(* IEC 61131-3 sources: CODESYS-IO-Visualization/CODESYS-IO-Visualization.fbsproj/Subs/IO, 10 files *)

(* ---- CodeSysCPU.prg.st ---- *)
PROGRAM CodeSysCPU

VAR_IN_OUT
	cpu: CodeSysCPU_UDT;
END_VAR

IF (cpu.PersistSize = 0) THEN
	cpu.PersistSize := SIZEOF(CodeSysCPU_UDT);
END_IF;

IF (cpu.Init OR cpu.AppResult <> 0) THEN
	cpu.App := AppGetCurrent(pResult := ADR(cpu.AppResult));
	IF (cpu.App <> 0) AND(cpu.AppResult = 0) THEN
		cpu.AppInfo := AppGetApplicationInfo(pApp := cpu.App, pResult := ADR(cpu.AppInfoResult));
		IF (cpu.AppInfo <> 0) AND (cpu.AppInfoResult = 0) THEN
 			cpu.AppProjectName := TO_WSTRING(cpu.AppInfo^.pstProjectName^);
 			cpu.AppAuthor := TO_WSTRING(cpu.AppInfo^.pstAuthor^);
 			cpu.AppVersion := TO_WSTRING(cpu.AppInfo^.pstVersion^);
 			cpu.AppDescription := TO_WSTRING(cpu.AppInfo^.pstDescription^);
 			cpu.AppProfile := TO_WSTRING(cpu.AppInfo^.pstProfile^);

			GetDateYear(Clock := DT_TO_DATE(cpu.AppInfo^.dtLastChanges), value => cpu.AppLastChange.Year);
			GetDateMonth(Clock := DT_TO_DATE(cpu.AppInfo^.dtLastChanges), value => cpu.AppLastChange.Month);
			GetDayOfMonth(Clock := DT_TO_DATE(cpu.AppInfo^.dtLastChanges), value => cpu.AppLastChange.Day);
			GetDTHour(Clock := cpu.AppInfo^.dtLastChanges, value => cpu.AppLastChange.Hour);
			GetDTMinute(Clock := cpu.AppInfo^.dtLastChanges, value => cpu.AppLastChange.Minute);
			GetDTSecond(Clock := cpu.AppInfo^.dtLastChanges, value => cpu.AppLastChange.Second);
			cpu.AppLastChange.DateTimeString := DateTimeStampToString(DateTimeStamp := cpu.AppLastChange);
		END_IF;
	END_IF;
	cpu.Init := FALSE;
END_IF;

CycleTime(value := cpu.CT);
cpu.SampleSeconds := cpu.SampleSeconds + cpu.CT.Sec;

// only read memory and cpu data every 10 seconds
IF (cpu.SampleSeconds < 10.0) THEN
	RETURN;
END_IF;

cpu.SampleSeconds := 0.0;

// Get CPU Info - Raspberry Pi ONLY - requires Shell Access enabled in /etc/codesyscontrol/CODESYSControl_User.cfg file
// Add
//	[SysProcess]
//  Command=AllowAll
ReadCPUDetails();

cpu.CpuUsage := ReadCPUDetails.cpuUsage;
cpu.Temperature := ReadCPUDetails.cpuTemp;
cpu.MemFree := ReadCPUDetails.memFree;
cpu.MemFree_MB := ReadCPUDetails.memFree_MB;
cpu.memTotal := ReadCPUDetails.memTotal;
cpu.memTotal_MB := ReadCPUDetails.memTotal_MB;
cpu.memUsed := ReadCPUDetails.memUsed;
cpu.memUsed_MB := ReadCPUDetails.memUsed_MB;

(* ---- IO_Simulator.prg.st ---- *)
__METADATA__
{
  "v3Meta": {
    "objectGuid": "030a1301-75cd-4f4e-867e-5d1ddb7f8ba8",
    "objectTypeGuid": "6f9dac99-8de1-4efc-8465-68ac443b7d08",
    "embeddedObjectTypeGuids": [
      "a9ed5b7e-75c5-4651-af16-d2c27e98cb94",
      "3b83b776-fb25-43b8-99f2-3c507c9143fc"
    ],
    "properties": {},
    "subObjects": {}
  }
}
__DECLARATION__
PROGRAM IO_Simulator
VAR_IN_OUT
	Data: IO_Simulator_UDT;
END_VAR
__IMPLEMENTATION__
Data.RandomNumber := OSCAT_BASIC.RDM(Data.RandomNumber);
Data.Noise := Data.RandomNumber * Data.irNoisePct;

Data.ChangeRamp(
	X := Data.irPercent,
	A_UP := Data.irChangeRate,
	A_DN := Data.irChangeRate * -1,
	VU_MAX := Data.irChangeRate,
	VD_MAX := Data.irChangeRate * -1,
	LIMIT_LOW := 0.0,
	LIMIT_HIGH := 100.0
);

IF (NOT Data.ibDisableOutput) THEN
	Data.orPercent := Data.Noise + Data.ChangeRamp.Y;
	Data.obValue := Data.ibValue;
END_IF;

Data.orValue := Data.irLowLimit + ((Data.orPercent / 100.0) * (Data.irHighLimit - Data.irLowLimit));

(* ---- IOA_Input.prg.st ---- *)
PROGRAM IOA_Input

VAR_IN_OUT
	Data: Channel_UDT;
END_VAR

VAR_INPUT
	ModuleStatus: DINT;
	ModuleCI: BOOL;
END_VAR

IF (Data.CI OR ModuleCI) THEN
	Data.StatusString := "Control Inhibited";
	Data.StatusCode := -1;
ELSE
	IF (Data.SimulationEnable AND Simulation.SimulationEnable) THEN
		ModuleStatus := 0;
		Data.ValueStatus := 0;
		Data.StatusCode := Data.Simulator.odiStatusCode;
		Data.StatusString := Data.Simulator.osStatusCode;
	ELSE
		IF (ModuleStatus > 0) THEN
			Data.StatusCode := ModuleStatus;
			Data.StatusString := "Module Failed, check Module Status";
		ELSE
			Data.StatusCode := WORD_TO_DINT(Data.ValueStatus);
			IO_StatusCodeToString(Data := Data);
		END_IF;
	END_IF;
END_IF;

Data.Invalid.Value := (Data.StatusCode > 0);
AlarmDigital(alarm := Data.Invalid);

IF (NOT FPU.IsRealNaN(Data.ValueRawAnalog)) THEN
	IF (Data.ValueRawAnalog > (Data.ZeroRaw + (Data.SpanRaw * 1.04))) THEN
		Data.ValueRawAnalog := Data.ZeroRaw + Data.SpanRaw;
	END_IF;

	IF (Data.ValueRawAnalog < (Data.ZeroRaw - (Data.SpanRaw * 0.04))) THEN
		Data.ValueRawAnalog := Data.ZeroRaw;
	END_IF;
END_IF;

IF (NOT Data.CI) AND (NOT ModuleCI) THEN
	IF (Data.SimulationEnable AND Simulation.SimulationEnable) THEN
		IO_Simulator(Data := Data.Simulator);
		Data.ValueEu := Data.Simulator.orValue;
	ELSE
		IF (NOT FPU.IsRealNaN(Data.ValueRawAnalog)) THEN
			IF (Data.SpanRaw <> 0.0) THEN
				Data.ValueEu := Data.ZeroEu + (((Data.ValueRawAnalog - Data.ZeroRaw) / Data.SpanRaw) * Data.SpanEu);
			ELSE
				Data.ValueEu := 0.0;
			END_IF;
		ELSE
			Data.ValueEu := 0.0;
		END_IF;
	END_IF;
END_IF;

IF (NOT FPU.IsRealNaN(Data.ValueRawAnalog)) THEN
	IF (Data.SpanEu <> 0.0) THEN
		Data.ValuePct := ((Data.ValueEu - Data.ZeroEu) / Data.SpanEu) * 100.0;
		IF (Data.ValuePct > 100.0) THEN
			Data.ValuePct := 100.0;
		END_IF;
		IF (Data.ValuePct < 0.0) THEN
			Data.ValuePct := 0.0;
		END_IF;
	ELSE
		Data.ValuePct := 0.0;
	END_IF;
ELSE
	Data.ValuePct := 0.0;
END_IF;

(* ---- IOA_Output.prg.st ---- *)
PROGRAM IOA_Output

VAR_IN_OUT
	Data: Channel_UDT;
END_VAR

VAR_INPUT
	ModuleStatus: DINT;
	ModuleCI: BOOL;
END_VAR

IF (Data.CI OR ModuleCI) THEN
	Data.StatusString := "Control Inhibited";
	Data.StatusCode := -1;
ELSE
	IF (ModuleStatus  > 0) THEN
		Data.StatusCode := ModuleStatus;
		Data.StatusString := "Module Failed, check Module Status";
	ELSE
		Data.StatusCode := WORD_TO_DINT(Data.ValueStatus);
		IO_StatusCodeToString(Data := Data);
	END_IF;
END_IF;

Data.Invalid.Value := (Data.StatusCode > 0);
AlarmDigital(alarm := Data.Invalid);

IF (NOT Data.CI) AND (NOT ModuleCI) THEN
	IF (Data.SpanEu <> 0.0) THEN
		Data.ValueRawAnalogOut := Data.ZeroRaw + (((Data.ValueEu - Data.ZeroEu) / Data.SpanEu) * Data.SpanRaw);
	ELSE
		Data.ValueRawAnalogOut := 0.0;
	END_IF;

	IF (Data.ValueRawAnalogOut > (Data.ZeroRaw + (Data.SpanRaw * 1.04))) THEN
		Data.ValueRawAnalogOut := Data.ZeroRaw + Data.SpanRaw;
	END_IF;

	IF (Data.ValueRawAnalogOut < (Data.ZeroRaw - (Data.SpanRaw * 0.04))) THEN
		Data.ValueRawAnalogOut := Data.ZeroRaw;
	END_IF;
END_IF;

IF (Data.SpanEu <> 0.0) THEN
	Data.ValuePct := ((Data.ValueEu - Data.ZeroEu) / Data.SpanEu) * 100.0;
	IF (Data.ValuePct > 100.0) THEN
		Data.ValuePct := 100.0;
	END_IF;
	IF (Data.ValuePct < 0.0) THEN
		Data.ValuePct := 0.0;
	END_IF;
ELSE
	Data.ValuePct := 0.0;
END_IF;

(* ---- IOD_Input.prg.st ---- *)
PROGRAM IOD_Input

VAR_IN_OUT
	Data: Channel_UDT;
END_VAR

VAR_INPUT
	ModuleStatus: DINT;
	ModuleCI: BOOL;
END_VAR

IF (Data.CI OR ModuleCI) THEN
	Data.StatusString := "Control Inhibited";
	Data.StatusCode := -1;
ELSE
	IF (Data.SimulationEnable AND Simulation.SimulationEnable) THEN
		ModuleStatus := 0;
		Data.ValueStatus := 0;
		Data.StatusCode := Data.Simulator.odiStatusCode;
		Data.StatusString := Data.Simulator.osStatusCode;
	ELSE
		IF (ModuleStatus > 0) THEN
			Data.StatusCode := ModuleStatus;
			Data.StatusString := "Module Failed, check Module Status";
		ELSE
			Data.StatusCode := WORD_TO_DINT(Data.ValueStatus);
			IO_StatusCodeToString(Data := Data);
		END_IF;
	END_IF;
END_IF;

Data.Invalid.Value := (Data.StatusCode > 0);
AlarmDigital(alarm := Data.Invalid);

IF (NOT Data.CI) AND (NOT ModuleCI) THEN
	IF (Data.InvertValue) THEN
		IF (Data.SimulationEnable AND Simulation.SimulationEnable) THEN
			IO_Simulator(Data := Data.Simulator);
			Data.ValueDig := (NOT Data.Simulator.obValue);
		ELSE
			Data.ValueDig := (NOT Data.ValueRawDigital);
		END_IF;
	ELSE
		IF (Data.SimulationEnable AND Simulation.SimulationEnable) THEN
			IO_Simulator(Data := Data.Simulator);
			Data.ValueDig := Data.Simulator.obValue;
		ELSE
			Data.ValueDig := Data.ValueRawDigital;
		END_IF;
	END_IF;
END_IF;

(* ---- IOD_Output.prg.st ---- *)
PROGRAM IOD_Output

VAR_IN_OUT
	Data: Channel_UDT;
END_VAR

VAR_INPUT
	ModuleStatus: DINT;
	ModuleCI: BOOL;
END_VAR

IF (Data.CI OR ModuleCI) THEN
	Data.StatusString := "Control Inhibited";
	Data.StatusCode := -1;
ELSE
	IF (ModuleStatus > 0) THEN
		Data.StatusCode := ModuleStatus;
		Data.StatusString := "Module Failed, check Module Status";
	ELSE
		Data.StatusCode := WORD_TO_DINT(Data.ValueStatus);
		IO_StatusCodeToString(Data := Data);
	END_IF;
END_IF;

Data.Invalid.Value := (Data.StatusCode > 0);
AlarmDigital(alarm := Data.Invalid);

IF (NOT Data.CI) AND (NOT ModuleCI) THEN
	IF (Data.InvertValue) THEN
		Data.ValueRawDigitalOut := (NOT Data.ValueDig);
	ELSE
		Data.ValueRawDigitalOut := Data.ValueDig;
	END_IF;
END_IF;

(* ---- ReadCPUDetails.prg.st ---- *)
PROGRAM ReadCPUDetails
VAR
	getTempCmd : STRING := 'vcgencmd measure_temp | sed $"s/temp=//; s/$'C//$"';
 	getCPUUsageCmd : STRING := 'top -bn1 | awk $'/^%Cpu/ {printf $"%.1f\n$", $$2}$'';
 	getMemoryTotalCmd : STRING := 'free | grep -E $"Mem$" | awk $'{print $$2}$'';
 	getMemoryUsedCmd : STRING := 'free | grep -E $"Mem$" | awk $'{print $$3}$'';
 	getMemoryFreeCmd : STRING := 'free | grep -E $"Mem$" | awk $'{print $$4}$'';

	command1 : STRING;
	commandToRun: INT;	// 0 = Temp, 1 = CPU, 2 = Memory Total, 3 = Memory Used, 4 = Memory Free

	stdout : STRING(1000) := '';
	Result : RTS_IEC_RESULT;
	xExecuteSysP: BOOL;
	xshowCPUInfo: BOOL;
	done: BOOL;

	dlyTimer: Timer_UDT := (PT := 0.25);
END_VAR

VAR_OUTPUT
	cpuTemp: REAL;
	cpuUsage: REAL;
	memTotal: DINT;
	memTotal_MB: REAL;
	memUsed: DINT;
	memUsed_MB: REAL;
	memFree: DINT;
	memFree_MB: REAL;
END_VAR

//Attention: allow shell commands in CODESYSControl.cfg

CASE commandToRun OF
	0: command1 := getTempCmd;
	1: command1 := getCPUUsageCmd;
	2: command1 := getMemoryTotalCmd;
	3: command1 := getMemoryUsedCmd;
	4: command1 := getMemoryFreeCmd;
END_CASE;

dlyTimer.In := (NOT done);

Timer(TimerData := dlyTimer);

IF (dlyTimer.Q) THEN
	SysProcess.SysProcessExecuteCommand2(pszCommand:=command1, pszStdOut:=stdout, udiStdOutLen:= SIZEOF(stdout),pResult := ADR(Result));
	done := TRUE;
END_IF;

IF (done AND Result = CmpErrors.Errors.ERR_OK) THEN
	IF (LEN(stdout) > 0) THEN
		CASE commandToRun OF
			0: cpuTemp := STRING_TO_REAL(stdout);
			1: cpuUsage := STRING_TO_REAL(stdout);
			2: memTotal := STRING_TO_DINT(stdout);
			   memTotal_MB := DINT_TO_REAL(memTotal) / 1024.0;
			3: memUsed := STRING_TO_DINT(stdout);
			   memUsed_MB := DINT_TO_REAL(memUsed) / 1024.0;
			4: memFree := STRING_TO_DINT(stdout);
			   memFree_MB := DINT_TO_REAL(memFree) / 1024.0;
		END_CASE;
	END_IF;

	commandToRun := commandToRun + 1;
	IF (commandToRun > 4) THEN
		commandToRun := 0;
	END_IF;

	done := FALSE;
END_IF;

(* ---- RotorkValve.prg.st ---- *)
PROGRAM RotorkValve

VAR_IN_OUT
	Data: RotorkValve_UDT;
	InputData: RotorkValve_MBIO_InputData_UDT;
	OutputData: RotorkValve_MBIO_OutputData_UDT;
END_VAR

// Assign Input Data from either the Modbus Device or the Simulator
IF (Simulation.SimulationEnable AND Data.SimulationEnable) THEN
	RotorkValve_Simulator(Data := Data.Simulator);
	Data.InputData := Data.Simulator.InputData;
ELSE
	Data.InputData := InputData;
END_IF;

IF (NOT Data.CI) THEN
	// Output Data
	Data.OutputData.Reg05 := INT_TO_WORD(Data.Actuator_Control);
	Data.OutputData.Reg06 := REAL_TO_WORD(Data.Actuator_Position_Command * 10.0);
	Data.OutputData.Reg07 := INT_TO_WORD(Data.SignalLossAction);
	Data.OutputData.Reg13 := INT_TO_WORD(Data.SignalLossPosition);

	// Input Data
	Data.InputReg00 := Data.InputData.Reg00;
	Data.Actuator_Moving := Data.InputData.Reg00.0;
	Data.Valve_Closed := Data.InputData.Reg00.1;
	Data.Valve_Opened := Data.InputData.Reg00.2;
	Data.Running_Closed := Data.InputData.Reg00.3;
	Data.Running_Open := Data.InputData.Reg00.4;
	Data.Remote_Selected := Data.InputData.Reg00.5;
	Data.Local_Stop_Selected_Offline := Data.InputData.Reg00.6;
	Data.Local_Stop_Selected := Data.InputData.Reg00.7;
	Data.Thermostat_Tripped := Data.InputData.Reg00.8;
	Data.Monitor_Relay := Data.InputData.Reg00.9;
	Data.Valve_Obstructed := Data.InputData.Reg00.10;
	Data.Valve_Jammed := Data.InputData.Reg00.11;
	Data.Valve_Moving_By_Hand := Data.InputData.Reg00.12;
	Data.Moving_Inhibited_by_MIT := Data.InputData.Reg00.13;
	Data.Position_Control_Enabled := Data.InputData.Reg00.14;
	Data.EEPROM_Checksum_Failure := Data.InputData.Reg00.15;

	Data.InputReg01 := Data.InputData.Reg01;
	Data.Battery_Low := Data.InputData.Reg01.0;
	Data.Open_Interlock_Active := Data.InputData.Reg01.1;
	Data.Close_Interlock_Active := Data.InputData.Reg01.2;
	Data.DI_1 := Data.InputData.Reg01.3;
	Data.DI_2 := Data.InputData.Reg01.4;
	Data.DI_3 := Data.InputData.Reg01.5;
	Data.DI_4 := Data.InputData.Reg01.6;
	Data.Reserved_7 := Data.InputData.Reg01.7;
	Data.Reserved_8 := Data.InputData.Reg01.8;
	Data.Reserved_9 := Data.InputData.Reg01.9;
	Data.Control_Contention := Data.InputData.Reg01.10;
	Data.Partial_Stroke_Test_in_Progress := Data.InputData.Reg01.11;
	Data.Partial_Stroke_Test_Error := Data.InputData.Reg01.12;
	Data.General_Alarm := Data.InputData.Reg01.13;
	Data.Reserved_14 := Data.InputData.Reg01.14;
	Data.Reserved_15 := Data.InputData.Reg01.15;

	Data.Actuator_Torque := WORD_TO_REAL(Data.InputData.Reg02);
	Data.Valve_Position := WORD_TO_REAL(Data.InputData.Reg03) / 10.0;
	Data.Analog_Input := WORD_TO_REAL(Data.InputData.Reg04) / 10.0;

	// Modbus Slave Data
	Data.SlaveState := Data.InputData.State;
	Data.SlaveError := Data.InputData.Error;
	Data.SlaveErrorCode := Data.InputData.ErrorCode;

	IF (Data.SlaveState = 2) THEN
		Data.Status := INT_TO_DINT(Data.SlaveErrorCode);
	ELSE
		Data.Status := UINT_TO_DINT(Data.SlaveState) + 1000;
	END_IF;
ELSE
	Data.Status := DINT#-1;
END_IF

// Output Data
IF (Simulation.SimulationEnable AND Data.SimulationEnable) THEN
	Data.Simulator.OutputData := Data.OutputData;
ELSE
	OutputData := Data.OutputData;
END_IF;

(* ---- RotorkValve_Simulator.prg.st ---- *)
PROGRAM RotorkValve_Simulator

VAR_IN_OUT
	Data: RotorkValve_Simulator_UDT;
END_VAR

// Set Valve Data from ModbusIO
Data.ibUsePosCmd := TRUE;

// Check for Comm Fail and set the valve position based on SignalLoss settings
IF (Data.InputData.Error OR (Data.InputData.State <> 2) OR (Data.InputData.ErrorCode <> 0)) THEN
	CASE Data.OutputData.Reg07 OF
		1: Data.irPosCmd := 100.0;
		3: Data.irPosCmd := 0.0;
		5: Data.irPosCmd := Data.orPosition;
		7: Data.irPosCmd := WORD_TO_REAL(Data.OutputData.Reg13);
	END_CASE;
ELSE
	Data.irPosCmd := WORD_TO_REAL(Data.OutputData.Reg06) / 10.0;
END_IF;

Data.ibAlarm := Data.Battery_Low OR Data.Open_Interlock_Active OR Data.Close_Interlock_Active OR Data.General_Alarm;
Data.ibFault := Data.Thermostat_Tripped OR Data.Valve_Obstructed OR Data.Valve_Jammed OR Data.Moving_Inhibited_by_MIT OR Data.EEPROM_Checksum_Failure;

// Call Simulator
ValveSimulator(Data := Data);

// Set Valve Output information from simulator
Data.InputData.Reg02 := 55;
Data.InputData.Reg03 := REAL_TO_WORD(Data.orPosition * 10.0);
Data.InputData.Reg04 := REAL_TO_WORD(Data.Analog_Input * 10.0);

Data.InputData.Reg00.0 := (Data.PosCmd > (Data.ChangeRamp.Y + 0.05)) OR (Data.PosCmd < (Data.ChangeRamp.Y - 0.05)) ;
Data.InputData.Reg00.1 := Data.obClosed;
Data.InputData.Reg00.2 := Data.obOpened;
Data.InputData.Reg00.3 := Data.InputData.Reg00.0 AND (Data.PosCmd < (Data.ChangeRamp.Y - 0.05));
Data.InputData.Reg00.4 := Data.InputData.Reg00.0 AND (Data.PosCmd > (Data.ChangeRamp.Y + 0.05));
Data.InputData.Reg00.5 := Data.obRemote;
Data.InputData.Reg00.6 := (NOT Data.obRemote) AND (NOT Data.InputData.Reg00.0);
Data.InputData.Reg00.7 := (NOT Data.obRemote) AND (NOT Data.InputData.Reg00.0);
Data.InputData.Reg00.8 := Data.Thermostat_Tripped;
Data.InputData.Reg00.9 := Data.Monitor_Relay;
Data.InputData.Reg00.10 := Data.Valve_Obstructed;
Data.InputData.Reg00.11 := Data.Valve_Jammed;
Data.InputData.Reg00.12 := Data.Valve_Moving_By_Hand;
Data.InputData.Reg00.13 := Data.Moving_Inhibited_by_MIT;
Data.InputData.Reg00.14 := Data.Postion_Control_Enabled;
Data.InputData.Reg00.15 := Data.EEPROM_Checksum_Failure;

Data.InputData.Reg01.0 := Data.Battery_Low;
Data.InputData.Reg01.1 := Data.Open_Interlock_Active;
Data.InputData.Reg01.2 := Data.Close_Interlock_Active;
Data.InputData.Reg01.3 := Data.DI_1;
Data.InputData.Reg01.4 := Data.DI_2;
Data.InputData.Reg01.5 := Data.DI_3;
Data.InputData.Reg01.6 := Data.DI_4;
Data.InputData.Reg01.7 := Data.Reserved_7;
Data.InputData.Reg01.8 := Data.Reserved_8;
Data.InputData.Reg01.9 := Data.Reserved_9;
Data.InputData.Reg01.10 := Data.Control_Contention;
Data.InputData.Reg01.11 := Data.Partial_Stroke_Test_in_Progress;
Data.InputData.Reg01.12 := Data.Partial_Stroke_Test_Error;
Data.InputData.Reg01.13 := Data.General_Alarm;
Data.InputData.Reg01.14 := Data.Reserved_14;
Data.InputData.Reg01.15 := Data.Reserved_15;

(* ---- ValveSimulator.prg.st ---- *)
__METADATA__
{
  "v3Meta": {
    "objectGuid": "ac6a8131-c4c6-4e28-ac6c-b30390678bef",
    "objectTypeGuid": "6f9dac99-8de1-4efc-8465-68ac443b7d08",
    "embeddedObjectTypeGuids": [
      "a9ed5b7e-75c5-4651-af16-d2c27e98cb94",
      "3b83b776-fb25-43b8-99f2-3c507c9143fc"
    ],
    "properties": {},
    "subObjects": {}
  }
}
__DECLARATION__
PROGRAM ValveSimulator

VAR_IN_OUT
	Data: ValveSimulator_UDT;
END_VAR

VAR
END_VAR
__IMPLEMENTATION__
Data.RandomNumber := OSCAT_BASIC.RDM(Data.RandomNumber);

IF (NOT Data.obClosed) AND (NOT Data.obOpened) THEN
	Data.Noise := Data.RandomNumber * Data.irNoisePct;
ELSE
	Data.Noise := 0.0;
END_IF;

Data.CoastTimer(
	IN := (NOT Data.ibOpenCmd) AND (NOT Data.ibCloseCmd),
	PT := REAL_TO_TIME(Data.irCoastTime * 1000.0)
);

IF (Data.ibAuto AND (NOT Data.ibDisableCommands)) THEN
	IF (Data.ibUsePosCmd) THEN
		Data.PosCmd := Data.irPosCmd;
	ELSE
		IF (Data.ibOpenCmd) AND (NOT Data.ibCloseCmd) THEN
			Data.PosCmd := 100.0;
		END_IF;

		IF (Data.ibCloseCmd) AND (NOT Data.ibOpenCmd) THEN
			Data.PosCmd := 0.0;
		END_IF;

		IF Data.CoastTimer.Q THEN
			Data.PosCmd := Data.orPosition;
		END_IF;
	END_IF;
END_IF;

Data.ChangeRamp(
	X := Data.PosCmd,
	A_UP := Data.irChangeRate,
	A_DN := Data.irChangeRate * -1,
	VU_MAX := Data.irChangeRate,
	VD_MAX := Data.irChangeRate * -1,
	LIMIT_LOW := 0.0,
	LIMIT_HIGH := 100.0
);

Data.orPosition := Data.Noise + Data.ChangeRamp.Y;

Data.obClosed := (Data.orPosition < Data.irClosedPct);
Data.obOpened := (Data.orPosition > Data.irOpenedPct);
Data.obRemote := Data.ibAuto;
Data.obFailed := Data.ibFault;
Data.obAlarm := Data.ibAlarm;
